(* Logix 5000 project; controller AdvManLab vendor 1 type 14 code 158 rev 28.12; software revision 28.01; part 8 of 13 *)
(* tags used below, declared in another part *)
   Counter_1 : COUNTER;
   Advance_Slide : BOOL;
   Auto_Valves01 : SINT;
   Auto_Valves02 : SINT;
   C1HoldBack : PalletStop;
   C1RobotStop : PalletStop;
   C23Diverter : PalletStop;
   C23DivHoldBack : PalletStop;
   C2HoldBack : PalletStop;
   C2RobotStop : PalletStop;
   C31DiverterHoldBack : PalletStop;
   C3RobotStop : PalletStop;
   CNC4Bools : DINT;
   CNC_4_ProgToRun : DINT;
   Empty_pallet : BOOL;
   Extend_Stop : BOOL;
   FaultReset : BOOL;
   Festo_Air_On : BOOL;
   Fetching_matl : BOOL;
   FromCNC4 : CNC_Datablock;   // Data From CNC4
   Gantry_busy : BOOL;
   Gantry_prep : BOOL;
   Gantry_reload : BOOL;
   Gantry_start : BOOL;
   Holding_matl : BOOL;
   Lower_Slide : BOOL;
   Man_Valves : DINT[8];
   Man_Valves01 : SINT;
   Man_Valves02 : SINT;
   Matl_delivered : BOOL;
   ONS : DINT;
   Part_dropped : BOOL;
   Part_from_conv_holding : BOOL;
   Part_ready_for_Gantry : BOOL;
   Picking_up_part : BOOL;
   Raise_Slide : BOOL;
   Return_Slide : BOOL;
   RFIDTP4 : ALIAS FOR RFID_N055:I.Channel[1].TagPresent;   // RFID Tag at Cell C23 Hold Back Stop
   Run_gantry_logic : BOOL;
   RunPartOnCNC4 : BOOL;
   TimerG1 : TIMER;
   TimerG2 : TIMER;
   TimerG3 : TIMER;
   TimerG4 : TIMER;
   TimerG5 : TIMER;
   TimerG6 : TIMER;
   TimerG7 : TIMER;
   TimerG8 : TIMER;
   ToCNC4 : CNC_Datablock;   // Data To CNC4
   Vac_On : BOOL;
(* MainProgram, continued *)

ROUTINE CNC4   (* ladder *)
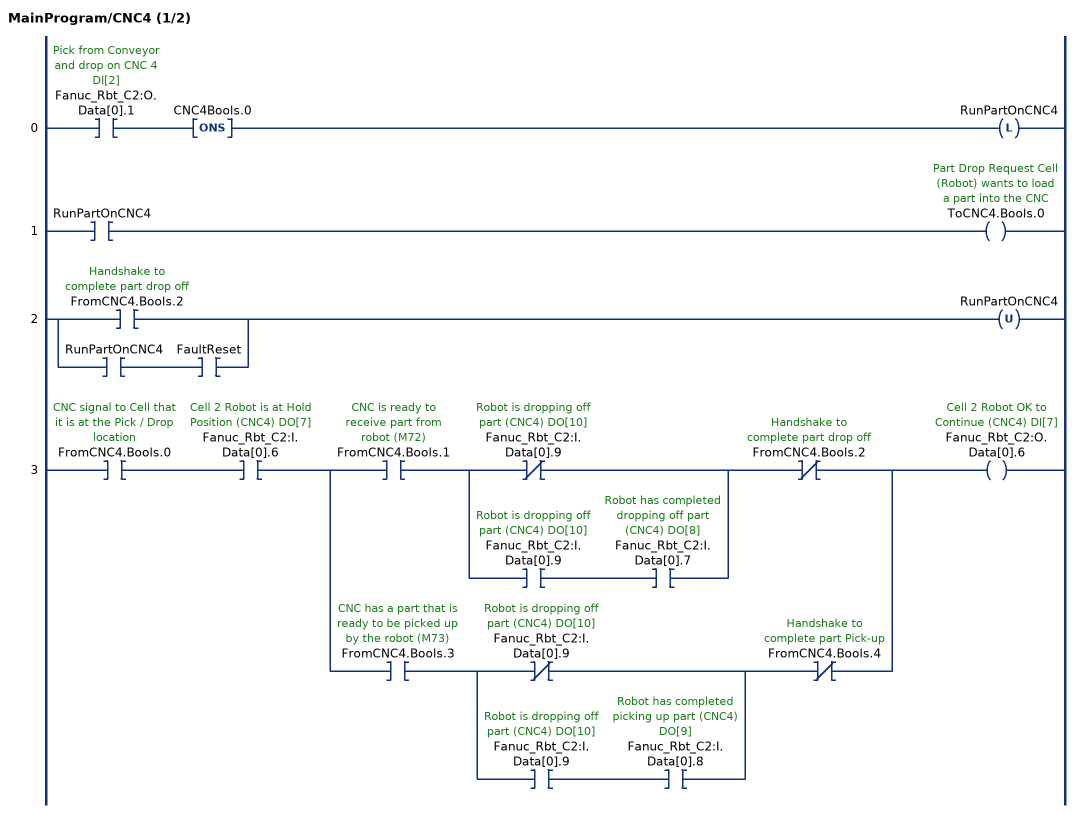
   0: XIC(Fanuc_Rbt_C2:O.Data[0].1)ONS(CNC4Bools.0)OTL(RunPartOnCNC4);
   1: XIC(RunPartOnCNC4)OTE(ToCNC4.Bools.0);
   2: [XIC(FromCNC4.Bools.2) ,XIC(RunPartOnCNC4) XIC(FaultReset) ]OTU(RunPartOnCNC4);
   3: XIC(FromCNC4.Bools.0)XIC(Fanuc_Rbt_C2:I.Data[0].6)[XIC(FromCNC4.Bools.1) [XIO(Fanuc_Rbt_C2:I.Data[0].9) ,XIC(Fanuc_Rbt_C2:I.Data[0].9) XIC(Fanuc_Rbt_C2:I.Data[0].7) ] XIO(FromCNC4.Bools.2) ,XIC(FromCNC4.Bools.3) [XIO(Fanuc_Rbt_C2:I.Data[0].9) ,XIC(Fanuc_Rbt_C2:I.Data[0].9) XIC(Fanuc_Rbt_C2:I.Data[0].8) ] XIO(FromCNC4.Bools.4) ]OTE(Fanuc_Rbt_C2:O.Data[0].6);
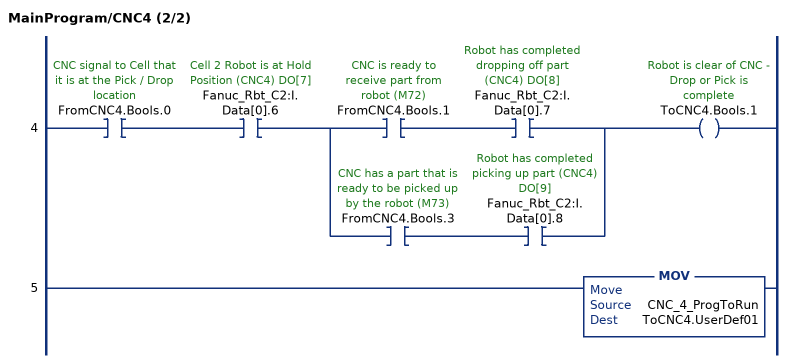
   4: XIC(FromCNC4.Bools.0)XIC(Fanuc_Rbt_C2:I.Data[0].6)[XIC(FromCNC4.Bools.1) XIC(Fanuc_Rbt_C2:I.Data[0].7) ,XIC(FromCNC4.Bools.3) XIC(Fanuc_Rbt_C2:I.Data[0].8) ]OTE(ToCNC4.Bools.1);
   5: MOV(CNC_4_ProgToRun,ToCNC4.UserDef01);
END_ROUTINE

ROUTINE Control_Valve   (* ladder *)
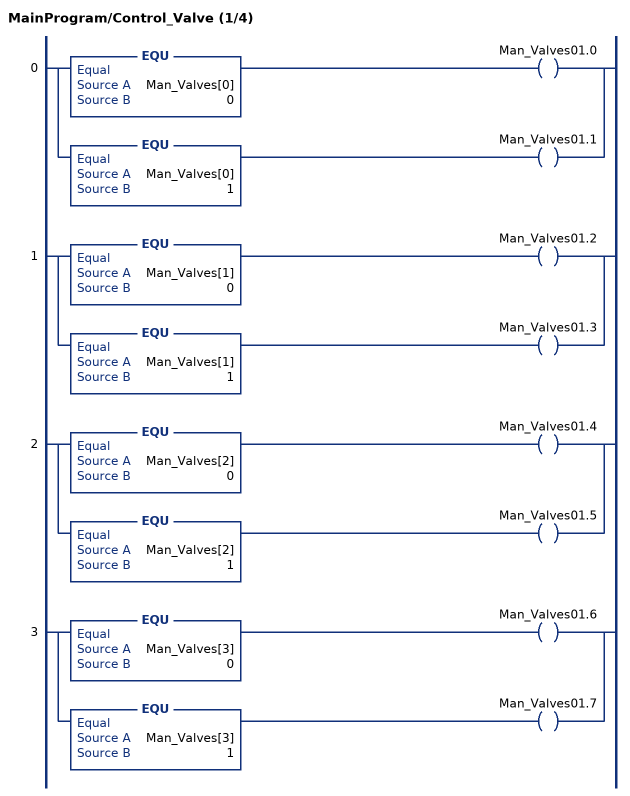
   0: [EQU(Man_Valves[0],0) OTE(Man_Valves01.0) ,EQU(Man_Valves[0],1) OTE(Man_Valves01.1) ];
   1: [EQU(Man_Valves[1],0) OTE(Man_Valves01.2) ,EQU(Man_Valves[1],1) OTE(Man_Valves01.3) ];
   2: [EQU(Man_Valves[2],0) OTE(Man_Valves01.4) ,EQU(Man_Valves[2],1) OTE(Man_Valves01.5) ];
   3: [EQU(Man_Valves[3],0) OTE(Man_Valves01.6) ,EQU(Man_Valves[3],1) OTE(Man_Valves01.7) ];
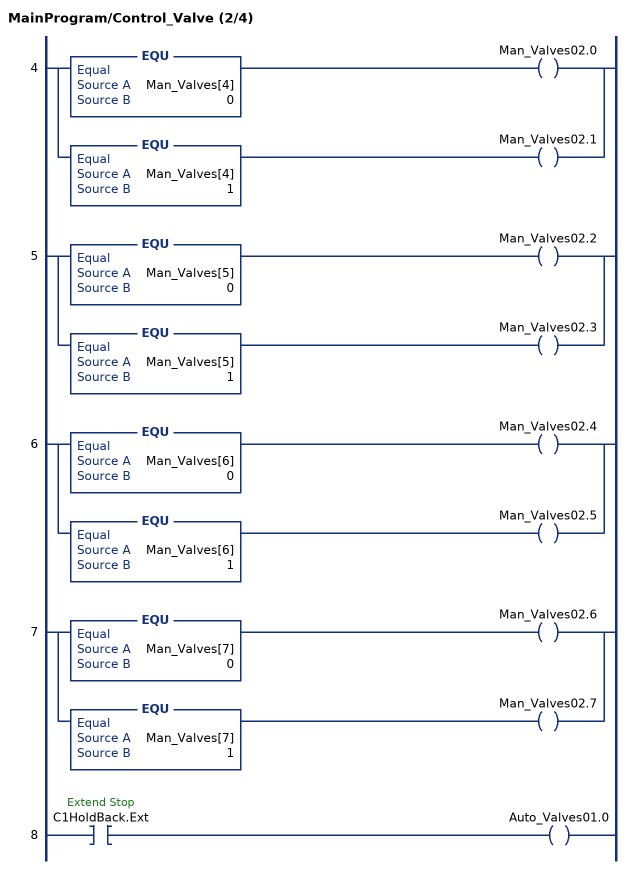
   4: [EQU(Man_Valves[4],0) OTE(Man_Valves02.0) ,EQU(Man_Valves[4],1) OTE(Man_Valves02.1) ];
   5: [EQU(Man_Valves[5],0) OTE(Man_Valves02.2) ,EQU(Man_Valves[5],1) OTE(Man_Valves02.3) ];
   6: [EQU(Man_Valves[6],0) OTE(Man_Valves02.4) ,EQU(Man_Valves[6],1) OTE(Man_Valves02.5) ];
   7: [EQU(Man_Valves[7],0) OTE(Man_Valves02.6) ,EQU(Man_Valves[7],1) OTE(Man_Valves02.7) ];
   8: XIC(C1HoldBack.Ext)OTE(Auto_Valves01.0);
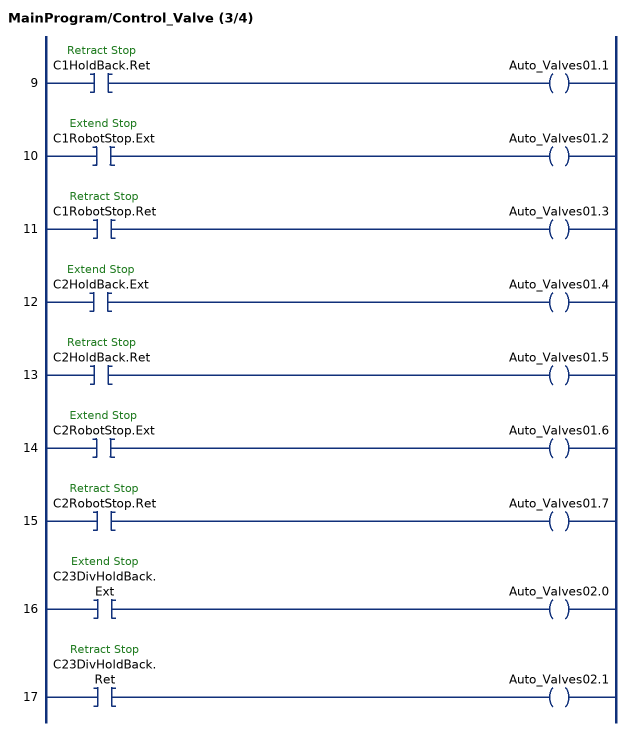
   9: XIC(C1HoldBack.Ret)OTE(Auto_Valves01.1);
   10: XIC(C1RobotStop.Ext)OTE(Auto_Valves01.2);
   11: XIC(C1RobotStop.Ret)OTE(Auto_Valves01.3);
   12: XIC(C2HoldBack.Ext)OTE(Auto_Valves01.4);
   13: XIC(C2HoldBack.Ret)OTE(Auto_Valves01.5);
   14: XIC(C2RobotStop.Ext)OTE(Auto_Valves01.6);
   15: XIC(C2RobotStop.Ret)OTE(Auto_Valves01.7);
   16: XIC(C23DivHoldBack.Ext)OTE(Auto_Valves02.0);
   17: XIC(C23DivHoldBack.Ret)OTE(Auto_Valves02.1);
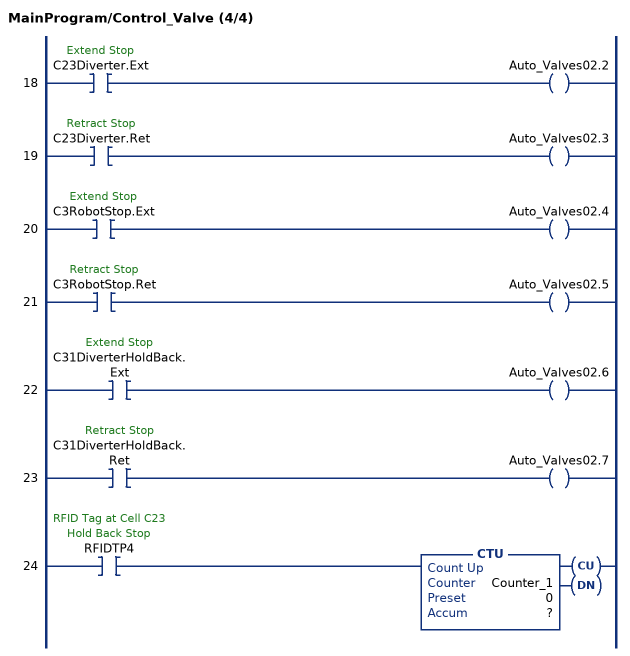
   18: XIC(C23Diverter.Ext)OTE(Auto_Valves02.2);
   19: XIC(C23Diverter.Ret)OTE(Auto_Valves02.3);
   20: XIC(C3RobotStop.Ext)OTE(Auto_Valves02.4);
   21: XIC(C3RobotStop.Ret)OTE(Auto_Valves02.5);
   22: XIC(C31DiverterHoldBack.Ext)OTE(Auto_Valves02.6);
   23: XIC(C31DiverterHoldBack.Ret)OTE(Auto_Valves02.7);
   24: XIC(RFIDTP4)CTU(Counter_1,?,?);
END_ROUTINE

ROUTINE Gantry_Logic_1   (* ladder *)
// Control pick and place
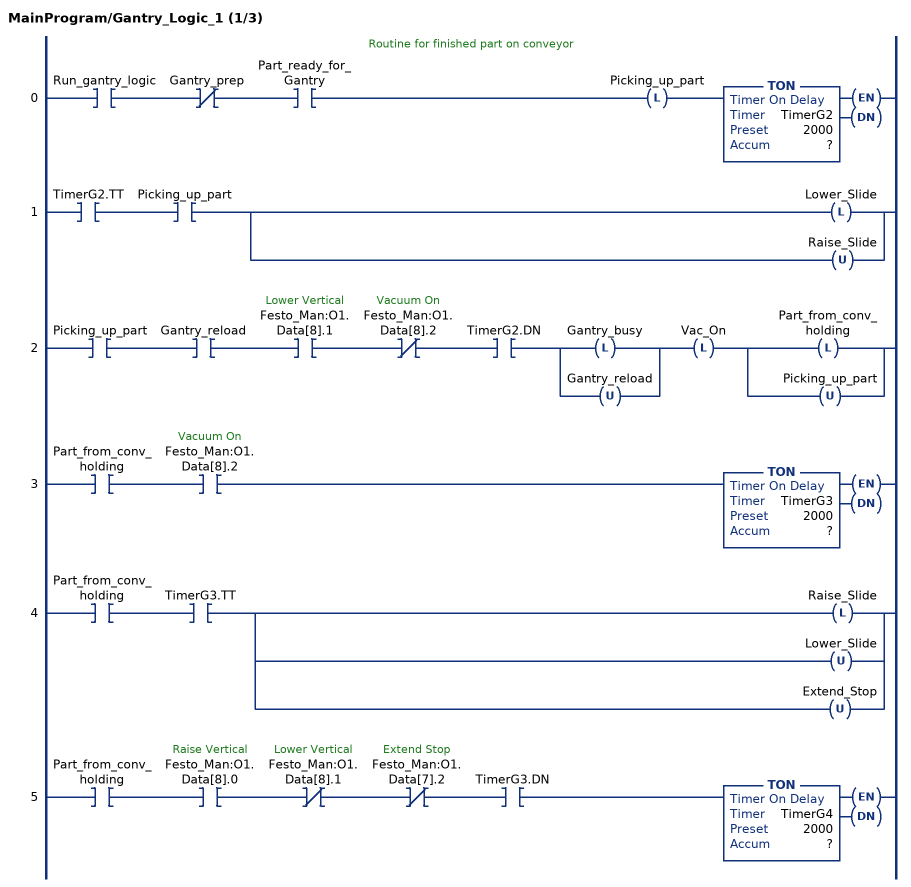
   // Routine for finished part on conveyor
   0: XIC(Run_gantry_logic)XIO(Gantry_prep)XIC(Part_ready_for_Gantry)OTL(Picking_up_part)TON(TimerG2,?,?);
   1: XIC(TimerG2.TT)XIC(Picking_up_part)[OTL(Lower_Slide) ,OTU(Raise_Slide) ];
   2: XIC(Picking_up_part)XIC(Gantry_reload)XIC(Festo_Man:O1.Data[8].1)XIO(Festo_Man:O1.Data[8].2)XIC(TimerG2.DN)[OTL(Gantry_busy) ,OTU(Gantry_reload) ]OTL(Vac_On)[OTL(Part_from_conv_holding) ,OTU(Picking_up_part) ];
   3: XIC(Part_from_conv_holding)XIC(Festo_Man:O1.Data[8].2)TON(TimerG3,?,?);
   4: XIC(Part_from_conv_holding)XIC(TimerG3.TT)[OTL(Raise_Slide) ,OTU(Lower_Slide) ,OTU(Extend_Stop) ];
   5: XIC(Part_from_conv_holding)XIC(Festo_Man:O1.Data[8].0)XIO(Festo_Man:O1.Data[8].1)XIO(Festo_Man:O1.Data[7].2)XIC(TimerG3.DN)TON(TimerG4,?,?);
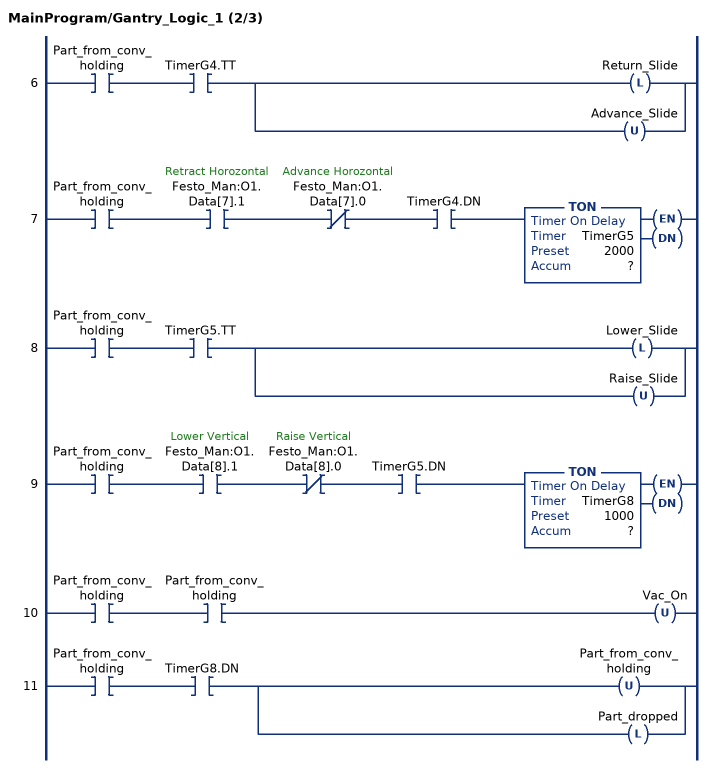
   6: XIC(Part_from_conv_holding)XIC(TimerG4.TT)[OTL(Return_Slide) ,OTU(Advance_Slide) ];
   7: XIC(Part_from_conv_holding)XIC(Festo_Man:O1.Data[7].1)XIO(Festo_Man:O1.Data[7].0)XIC(TimerG4.DN)TON(TimerG5,?,?);
   8: XIC(Part_from_conv_holding)XIC(TimerG5.TT)[OTL(Lower_Slide) ,OTU(Raise_Slide) ];
   9: XIC(Part_from_conv_holding)XIC(Festo_Man:O1.Data[8].1)XIO(Festo_Man:O1.Data[8].0)XIC(TimerG5.DN)TON(TimerG8,?,?);
   10: XIC(Part_from_conv_holding)XIC(Part_from_conv_holding)OTU(Vac_On);
   11: XIC(Part_from_conv_holding)XIC(TimerG8.DN)[OTU(Part_from_conv_holding) ,OTL(Part_dropped) ];
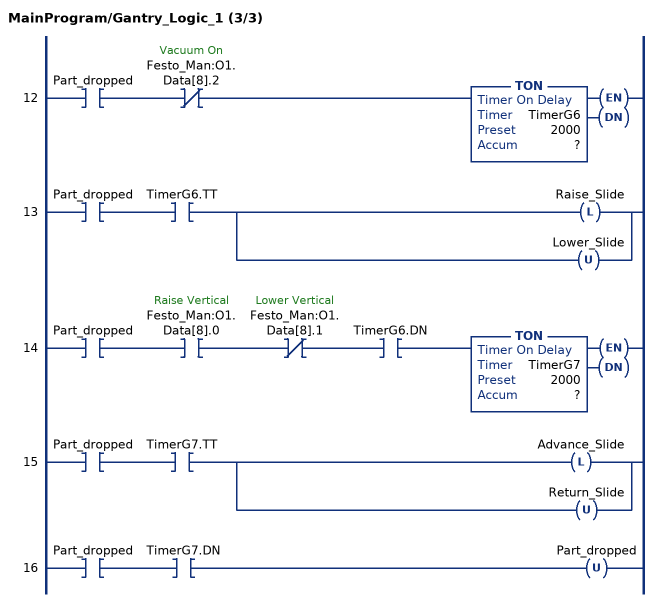
   12: XIC(Part_dropped)XIO(Festo_Man:O1.Data[8].2)TON(TimerG6,?,?);
   13: XIC(Part_dropped)XIC(TimerG6.TT)[OTL(Raise_Slide) ,OTU(Lower_Slide) ];
   14: XIC(Part_dropped)XIC(Festo_Man:O1.Data[8].0)XIO(Festo_Man:O1.Data[8].1)XIC(TimerG6.DN)TON(TimerG7,?,?);
   15: XIC(Part_dropped)XIC(TimerG7.TT)[OTL(Advance_Slide) ,OTU(Return_Slide) ];
   16: XIC(Part_dropped)XIC(TimerG7.DN)OTU(Part_dropped);
END_ROUTINE

ROUTINE Gantry_Logic_2   (* ladder *)
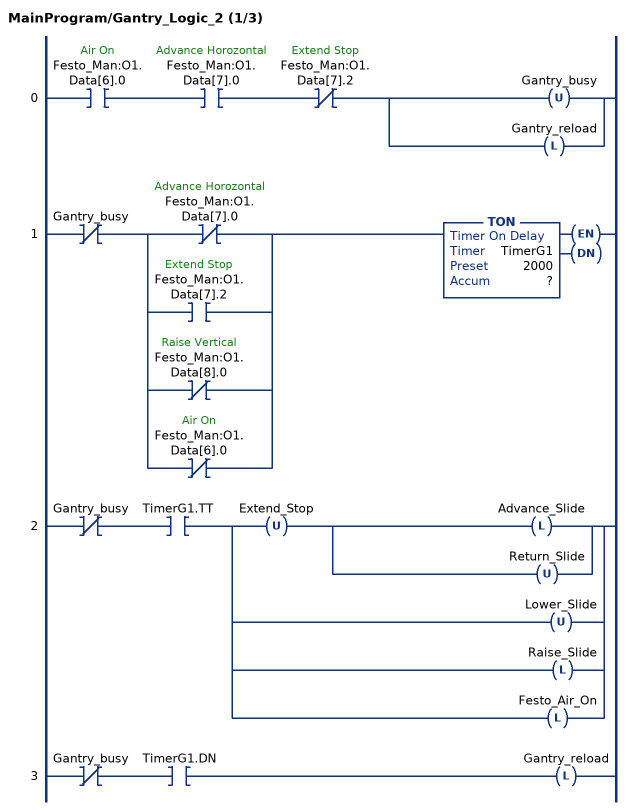
   0: XIC(Festo_Man:O1.Data[6].0)XIC(Festo_Man:O1.Data[7].0)XIO(Festo_Man:O1.Data[7].2)[OTU(Gantry_busy) ,OTL(Gantry_reload) ];
   1: XIO(Gantry_busy)[[XIO(Festo_Man:O1.Data[7].0) ,XIC(Festo_Man:O1.Data[7].2) ] ,XIO(Festo_Man:O1.Data[8].0) ,XIO(Festo_Man:O1.Data[6].0) ]TON(TimerG1,?,?);
   2: XIO(Gantry_busy)XIC(TimerG1.TT)[OTU(Extend_Stop) [OTL(Advance_Slide) ,OTU(Return_Slide) ] ,[OTU(Lower_Slide) ,OTL(Raise_Slide) ] ,OTL(Festo_Air_On) ];
   3: XIO(Gantry_busy)XIC(TimerG1.DN)OTL(Gantry_reload);
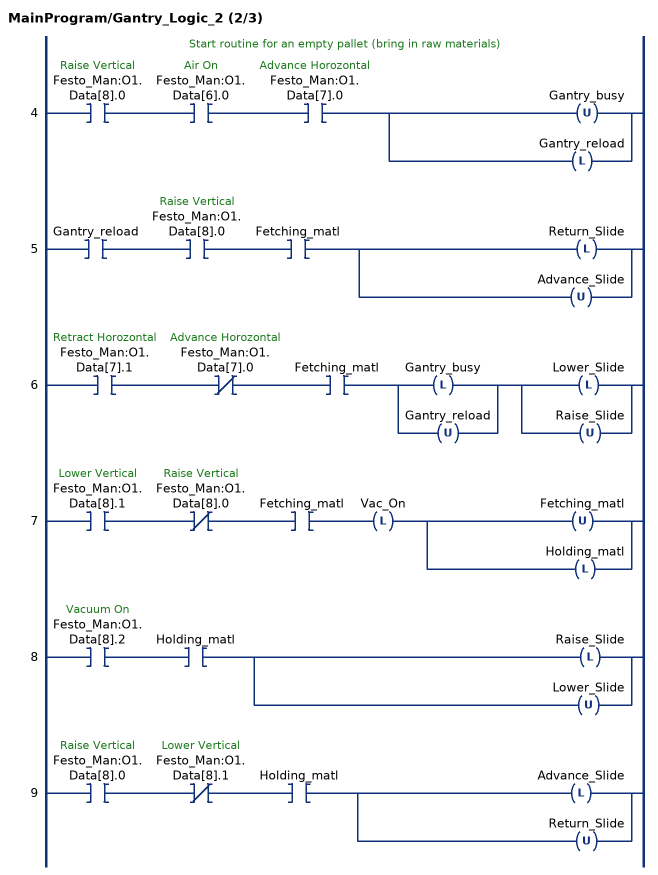
   // Start routine for an empty pallet (bring in raw materials)
   4: XIC(Festo_Man:O1.Data[8].0)XIC(Festo_Man:O1.Data[6].0)XIC(Festo_Man:O1.Data[7].0)[OTU(Gantry_busy) ,OTL(Gantry_reload) ];
   5: XIC(Gantry_reload)XIC(Festo_Man:O1.Data[8].0)XIC(Fetching_matl)[OTL(Return_Slide) ,OTU(Advance_Slide) ];
   6: XIC(Festo_Man:O1.Data[7].1)XIO(Festo_Man:O1.Data[7].0)XIC(Fetching_matl)[OTL(Gantry_busy) ,OTU(Gantry_reload) ][OTL(Lower_Slide) ,OTU(Raise_Slide) ];
   7: XIC(Festo_Man:O1.Data[8].1)XIO(Festo_Man:O1.Data[8].0)XIC(Fetching_matl)OTL(Vac_On)[OTU(Fetching_matl) ,OTL(Holding_matl) ];
   8: XIC(Festo_Man:O1.Data[8].2)XIC(Holding_matl)[OTL(Raise_Slide) ,OTU(Lower_Slide) ];
   9: XIC(Festo_Man:O1.Data[8].0)XIO(Festo_Man:O1.Data[8].1)XIC(Holding_matl)[OTL(Advance_Slide) ,OTU(Return_Slide) ];
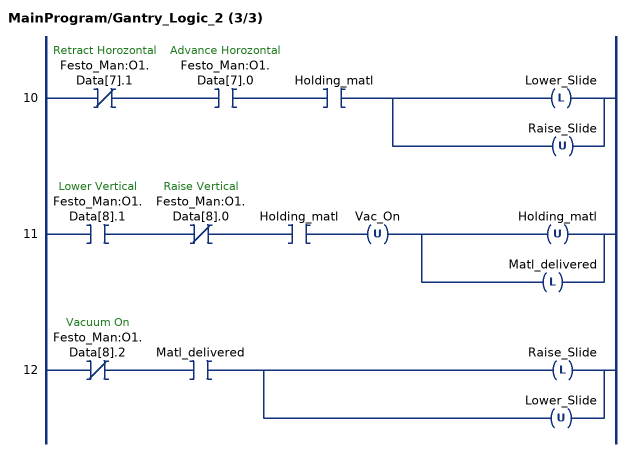
   10: XIO(Festo_Man:O1.Data[7].1)XIC(Festo_Man:O1.Data[7].0)XIC(Holding_matl)[OTL(Lower_Slide) ,OTU(Raise_Slide) ];
   11: XIC(Festo_Man:O1.Data[8].1)XIO(Festo_Man:O1.Data[8].0)XIC(Holding_matl)OTU(Vac_On)[OTU(Holding_matl) ,OTL(Matl_delivered) ];
   12: XIO(Festo_Man:O1.Data[8].2)XIC(Matl_delivered)[OTL(Raise_Slide) ,OTU(Lower_Slide) ];
END_ROUTINE

ROUTINE Gantry_Logic_Test   (* ladder *)
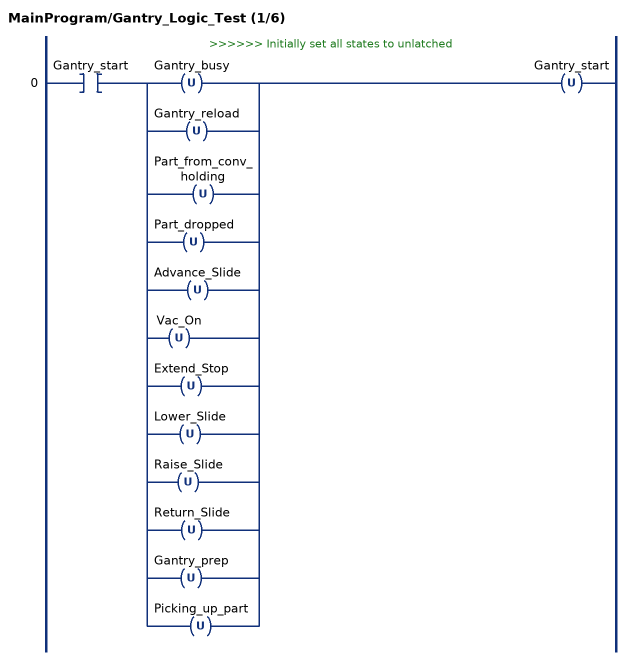
   // >>>>>> Initially set all states to unlatched
   0: XIC(Gantry_start)[OTU(Gantry_busy) ,OTU(Gantry_reload) ,OTU(Part_from_conv_holding) ,OTU(Part_dropped) ,OTU(Advance_Slide) ,OTU(Vac_On) ,OTU(Extend_Stop) ,OTU(Lower_Slide) ,OTU(Raise_Slide) ,OTU(Return_Slide) ,OTU(Gantry_prep) ,OTU(Picking_up_part) ]OTU(Gantry_start);
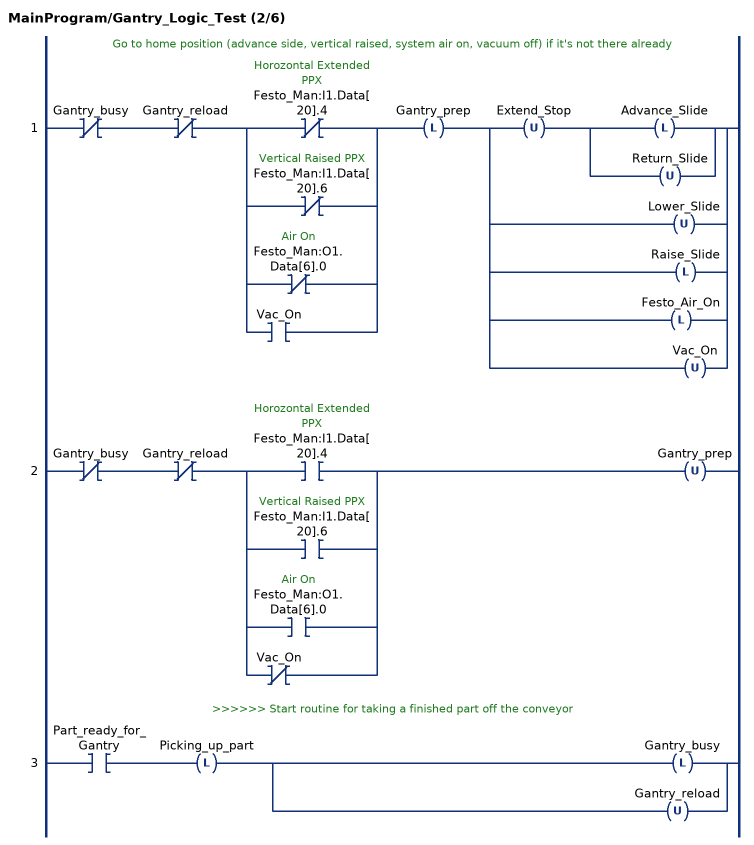
   // Go to home position (advance side, vertical raised, system air on, vacuum off) if it's not there already
   1: XIO(Gantry_busy)XIO(Gantry_reload)[XIO(Festo_Man:I1.Data[20].4) ,XIO(Festo_Man:I1.Data[20].6) ,XIO(Festo_Man:O1.Data[6].0) ,XIC(Vac_On) ]OTL(Gantry_prep)[OTU(Extend_Stop) [OTL(Advance_Slide) ,OTU(Return_Slide) ] ,[OTU(Lower_Slide) ,OTL(Raise_Slide) ] ,OTL(Festo_Air_On) ,OTU(Vac_On) ];
   2: XIO(Gantry_busy)XIO(Gantry_reload)[XIC(Festo_Man:I1.Data[20].4) ,XIC(Festo_Man:I1.Data[20].6) ,XIC(Festo_Man:O1.Data[6].0) ,XIO(Vac_On) ]OTU(Gantry_prep);
   // >>>>>> Start routine for taking a finished part off the conveyor
   3: XIC(Part_ready_for_Gantry)OTL(Picking_up_part)[OTL(Gantry_busy) ,OTU(Gantry_reload) ];
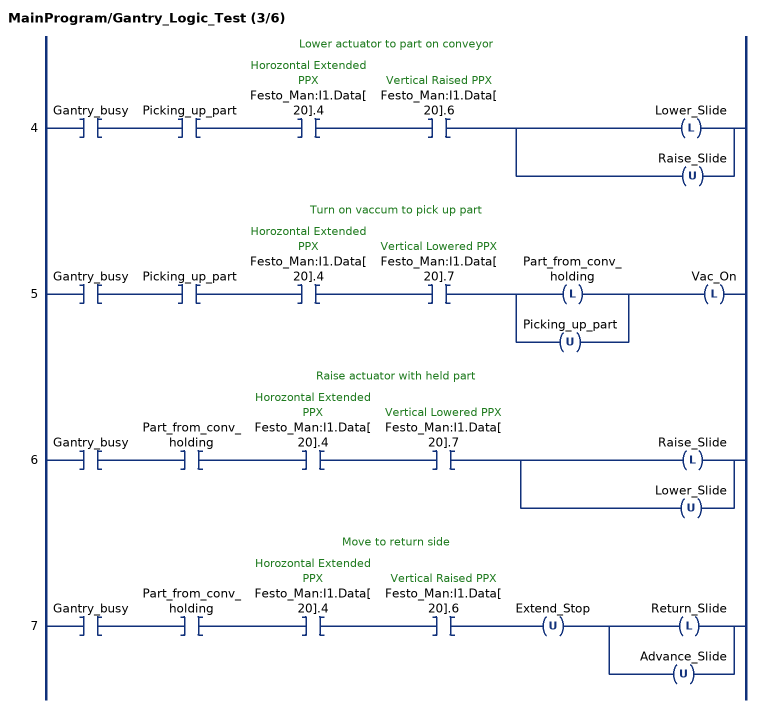
   // Lower actuator to part on conveyor
   4: XIC(Gantry_busy)XIC(Picking_up_part)XIC(Festo_Man:I1.Data[20].4)XIC(Festo_Man:I1.Data[20].6)[OTL(Lower_Slide) ,OTU(Raise_Slide) ];
   // Turn on vaccum to pick up part
   5: XIC(Gantry_busy)XIC(Picking_up_part)XIC(Festo_Man:I1.Data[20].4)XIC(Festo_Man:I1.Data[20].7)[OTL(Part_from_conv_holding) ,OTU(Picking_up_part) ]OTL(Vac_On);
   // Raise actuator with held part
   6: XIC(Gantry_busy)XIC(Part_from_conv_holding)XIC(Festo_Man:I1.Data[20].4)XIC(Festo_Man:I1.Data[20].7)[OTL(Raise_Slide) ,OTU(Lower_Slide) ];
   // Move to return side
   7: XIC(Gantry_busy)XIC(Part_from_conv_holding)XIC(Festo_Man:I1.Data[20].4)XIC(Festo_Man:I1.Data[20].6)OTU(Extend_Stop)[OTL(Return_Slide) ,OTU(Advance_Slide) ];
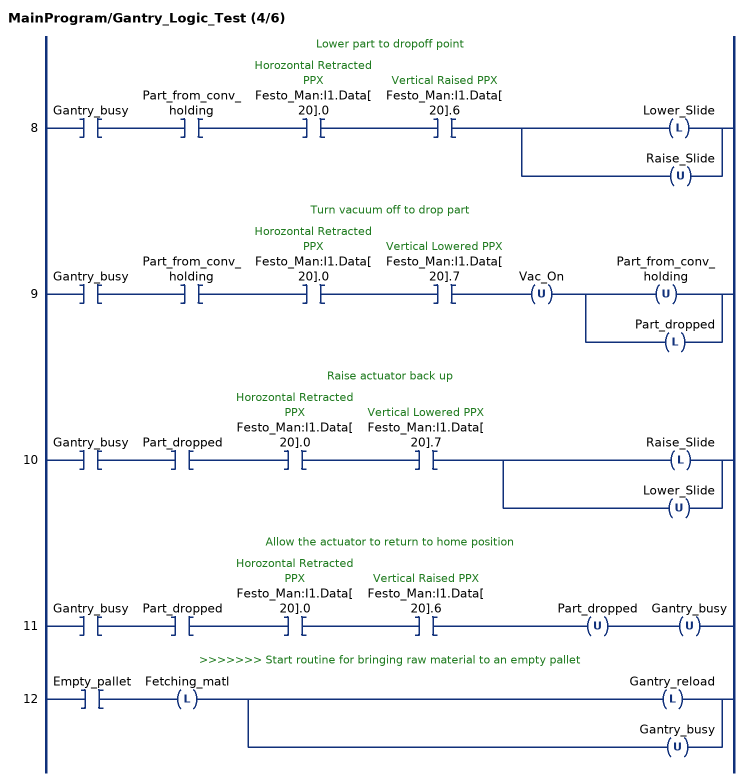
   // Lower part to dropoff point
   8: XIC(Gantry_busy)XIC(Part_from_conv_holding)XIC(Festo_Man:I1.Data[20].0)XIC(Festo_Man:I1.Data[20].6)[OTL(Lower_Slide) ,OTU(Raise_Slide) ];
   // Turn vacuum off to drop part
   9: XIC(Gantry_busy)XIC(Part_from_conv_holding)XIC(Festo_Man:I1.Data[20].0)XIC(Festo_Man:I1.Data[20].7)OTU(Vac_On)[OTU(Part_from_conv_holding) ,OTL(Part_dropped) ];
   // Raise actuator back up
   10: XIC(Gantry_busy)XIC(Part_dropped)XIC(Festo_Man:I1.Data[20].0)XIC(Festo_Man:I1.Data[20].7)[OTL(Raise_Slide) ,OTU(Lower_Slide) ];
   // Allow the actuator to return to home position
   11: XIC(Gantry_busy)XIC(Part_dropped)XIC(Festo_Man:I1.Data[20].0)XIC(Festo_Man:I1.Data[20].6)OTU(Part_dropped)OTU(Gantry_busy);
   // >>>>>>> Start routine for bringing raw material to an empty pallet
   12: XIC(Empty_pallet)OTL(Fetching_matl)[OTL(Gantry_reload) ,OTU(Gantry_busy) ];
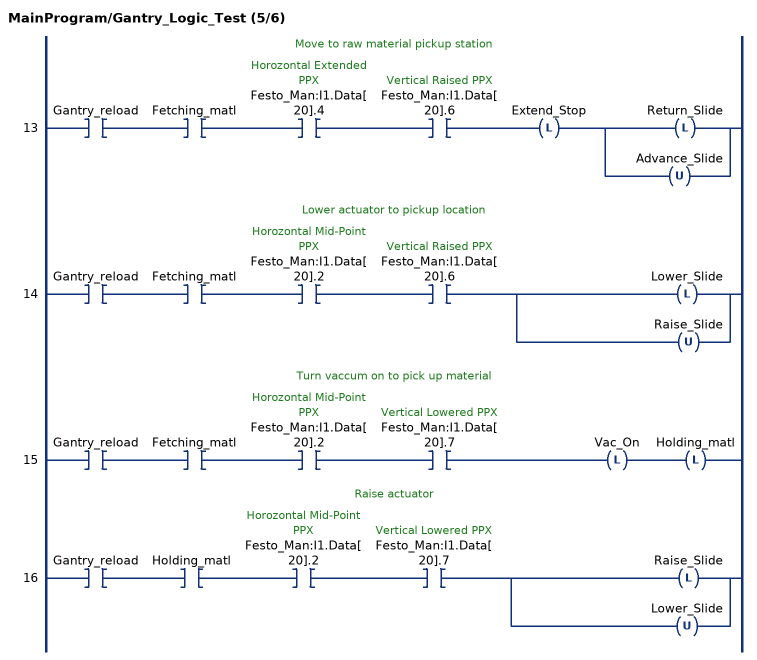
   // Move to raw material pickup station
   13: XIC(Gantry_reload)XIC(Fetching_matl)XIC(Festo_Man:I1.Data[20].4)XIC(Festo_Man:I1.Data[20].6)OTL(Extend_Stop)[OTL(Return_Slide) ,OTU(Advance_Slide) ];
   // Lower actuator to pickup location
   14: XIC(Gantry_reload)XIC(Fetching_matl)XIC(Festo_Man:I1.Data[20].2)XIC(Festo_Man:I1.Data[20].6)[OTL(Lower_Slide) ,OTU(Raise_Slide) ];
   // Turn vaccum on to pick up material
   15: XIC(Gantry_reload)XIC(Fetching_matl)XIC(Festo_Man:I1.Data[20].2)XIC(Festo_Man:I1.Data[20].7)OTL(Vac_On)OTL(Holding_matl);
   // Raise actuator
   16: XIC(Gantry_reload)XIC(Holding_matl)XIC(Festo_Man:I1.Data[20].2)XIC(Festo_Man:I1.Data[20].7)[OTL(Raise_Slide) ,OTU(Lower_Slide) ];
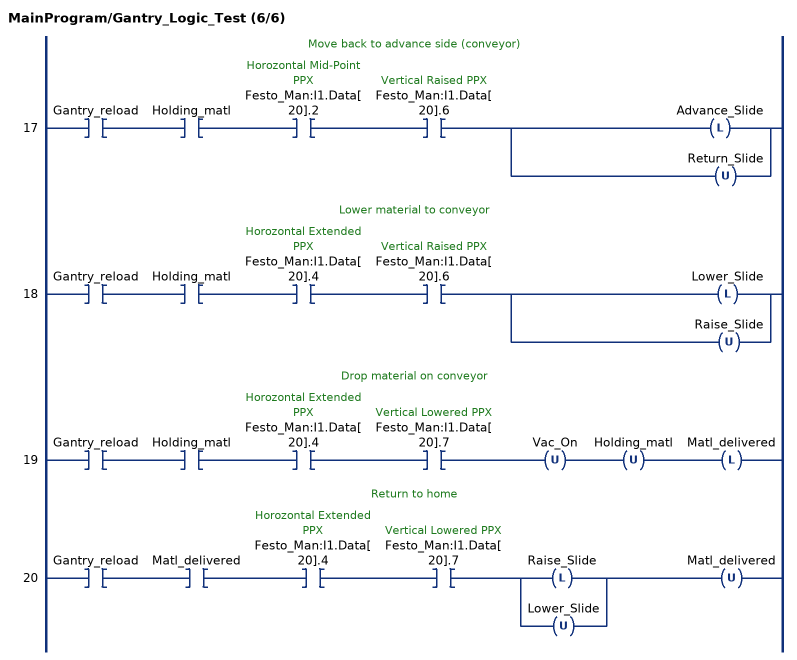
   // Move back to advance side (conveyor)
   17: XIC(Gantry_reload)XIC(Holding_matl)XIC(Festo_Man:I1.Data[20].2)XIC(Festo_Man:I1.Data[20].6)[OTL(Advance_Slide) ,OTU(Return_Slide) ];
   // Lower material to conveyor
   18: XIC(Gantry_reload)XIC(Holding_matl)XIC(Festo_Man:I1.Data[20].4)XIC(Festo_Man:I1.Data[20].6)[OTL(Lower_Slide) ,OTU(Raise_Slide) ];
   // Drop material on conveyor
   19: XIC(Gantry_reload)XIC(Holding_matl)XIC(Festo_Man:I1.Data[20].4)XIC(Festo_Man:I1.Data[20].7)OTU(Vac_On)OTU(Holding_matl)OTL(Matl_delivered);
   // Return to home
   20: XIC(Gantry_reload)XIC(Matl_delivered)XIC(Festo_Man:I1.Data[20].4)XIC(Festo_Man:I1.Data[20].7)[OTL(Raise_Slide) ,OTU(Lower_Slide) ]OTU(Matl_delivered);
END_ROUTINE
